// TIA Portal V18 export
DATA_BLOCK "!!nameOfDB$$"   // DB30, F_DB
{ S7_Optimized_Access := 'TRUE' }
   VAR
      AlwaysFALSE : Bool;
      AlwaysTRUE : Bool := TRUE;
      "!!ITERATOR_STRINGS$$" : Bool;
   END_VAR
BEGIN
END_DATA_BLOCK
